{attribute 'qualified_only'}
{attribute 'strict'}
{attribute 'conditionalshow'}
TYPE eSavePositionFile :
(
	{attribute 'hide'}
	ePostionHardDisk := 0,
	{attribute 'hide'}
	ePostionC := 1
);
END_TYPE

(* stored: Version 1.1.0.1, ProductVersion 3.1.4024.6
   DUT eSavePositionFile: Id {c7c9386a-bbe5-4950-87b9-c3e884b5a6d8} *)
